INTERFACE IHandling EXTENDS ZApplication.IUnit

END_INTERFACE

(* stored: Version 1.1.0.1
   Itf IHandling: Id {f4e7ca31-d9cc-4eaf-9168-2a6bfe22ea6e} *)
